FUNCTION_BLOCK AnalogInput_HMI (* Service Interface Function Block Type *)
  (* Standard: 61499-2 *)
  (* Version 0.0, 6/5/2026, Schneider Electric, template *)
  PACKAGE SE.Nereda;
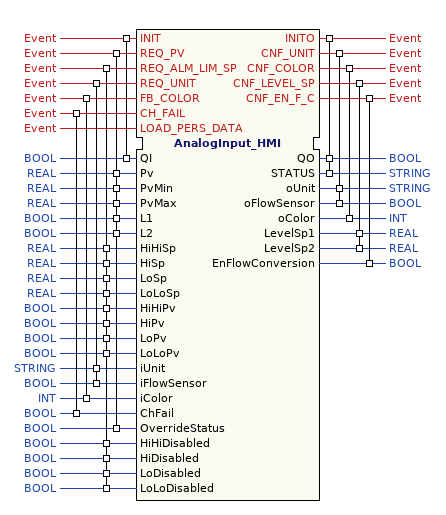
  EVENT_INPUT
    INIT WITH QI;
    REQ_PV WITH Pv, PvMin, PvMax, L1, L2, OverrideStatus;
    REQ_ALM_LIM_SP WITH HiHiSp, HiSp, LoSp, LoLoSp, HiHiPv, HiPv, LoPv, LoLoPv, HiHiDisabled, HiDisabled, LoDisabled, LoLoDisabled;
    REQ_UNIT WITH iUnit, iFlowSensor;
    FB_COLOR WITH iColor;
    CH_FAIL WITH ChFail;
    LOAD_PERS_DATA;
  END_EVENT
  EVENT_OUTPUT
    INITO WITH QO, STATUS;
    CNF_UNIT WITH oUnit, oFlowSensor;
    CNF_COLOR WITH oColor;
    CNF_LEVEL_SP WITH LevelSp1, LevelSp2;
    CNF_EN_F_C WITH EnFlowConversion;
  END_EVENT
  VAR_INPUT
    QI : BOOL;
    Pv : REAL;
    PvMin : REAL;
    PvMax : REAL;
    L1 : BOOL;
    L2 : BOOL;
    HiHiSp : REAL;
    HiSp : REAL;
    LoSp : REAL;
    LoLoSp : REAL;
    HiHiPv : BOOL;
    HiPv : BOOL;
    LoPv : BOOL;
    LoLoPv : BOOL;
    iUnit : STRING;
    iFlowSensor : BOOL;
    iColor : INT;
    ChFail : BOOL;
    OverrideStatus : BOOL;
    HiHiDisabled : BOOL;
    HiDisabled : BOOL;
    LoDisabled : BOOL;
    LoLoDisabled : BOOL;
  END_VAR
  VAR_OUTPUT
    QO : BOOL; (* Event Output Qualifier *)
    STATUS : STRING; (* Service Status *)
    oUnit : STRING;
    oFlowSensor : BOOL;
    oColor : INT;
    LevelSp1 : REAL;
    LevelSp2 : REAL;
    EnFlowConversion : BOOL; (* =1 ; Enable flow conversion from m3/s to m3/h *)
  END_VAR
  SERVICE /
    SEQUENCE 
    END_SEQUENCE
  END_SERVICE
END_FUNCTION_BLOCK
